// Filter messages, if already existing
FUNCTION F_Filter : BOOL
VAR_INPUT
	fbMessage:			FB_Message; // Input message
END_VAR
VAR
    nIndex:				UINT;	// Index counter
END_VAR

nIndex := 0;
WHILE nIndex < GVL.nBuffer DO
    IF GVL.aBuffer[nIndex].sDefault = fbMessage.sDefault THEN
        GVL.aBuffer[nIndex].bActive := TRUE;
        F_Filter := TRUE;
        RETURN;  // Message found
    END_IF
    nIndex := nIndex + 1;
END_WHILE

END_FUNCTION

(* stored: Version 1.1.0.1
   POU F_Filter: Id {e2511038-51cb-42c7-9bc5-a0c46a2fc45b}, SpecialFunc None *)
